PROGRAM P_Safety
VAR
END_VAR

END_PROGRAM

(* stored: Version 1.1.0.1, ProductVersion 3.1.4024.10
   POU P_Safety: Id {4a2af581-3054-4755-8b59-c878439b7ede}, SpecialFunc None *)
